FUNCTION_BLOCK StartIntervalCalc (* Basic Function Block Type *)
  (* Standard: 61499-2 *)
  (* Version 0.0, 7/5/2026, Schneider Electric, Template *)
  PACKAGE SE.Nereda;
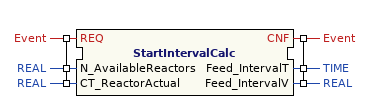
  EVENT_INPUT
    REQ WITH CT_ReactorActual, N_AvailableReactors; (* Normal Execution Request *)
  END_EVENT
  EVENT_OUTPUT
    CNF WITH Feed_IntervalT, Feed_IntervalV; (* Execution Confirmation *)
  END_EVENT
  VAR_INPUT
    N_AvailableReactors : REAL;
    CT_ReactorActual : REAL; (* Input event qualifier *)
  END_VAR
  VAR_OUTPUT
    Feed_IntervalT : TIME; (* Output event qualifier *)
    Feed_IntervalV : REAL;
  END_VAR
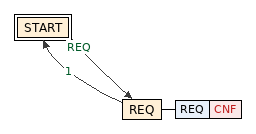
  EC_STATES
    START; (* Initial State *)
    REQ : REQ -> CNF; (* Normal execution *)
  END_STATES
  EC_TRANSITIONS
    START TO REQ := REQ;
    REQ TO START := 1;
  END_TRANSITIONS
  ALGORITHM REQ IN ST: (* Normally executed algorithm *)
;
IF N_AvailableReactors > 0.0 THEN
	Feed_IntervalV := CT_ReactorActual / N_AvailableReactors;
	Feed_IntervalT := REAL_TO_TIME(Feed_IntervalV);
ELSE
	Feed_IntervalV := 0;
	Feed_IntervalT := T#0s;
END_IF;
  END_ALGORITHM
END_FUNCTION_BLOCK
